// TIA Portal project "Rapid_Dyeing" (V16)
// Rapid machine for Dyeing Automation

(* hardware
DEVICE "HMI_1"  KTP400 Basic PN
   slot 0: "HMI_1"  KTP400 Basic PN  6AV2 123-2DB03-0AX0  16.0.0.0
   slot 1: "HMI_RT_1"  KTP400 Basic PN  6AV2 123-2DB03-0AX0  16.0.0.0
   slot 5: "HMI_1.IE_CP_1"  PROFINET Interface  16.0.0.0
      slot 1: "PROFINET Interface_1"  PROFINET Interface
         slot 1: "Port_1"  Port
DEVICE "S7-1200 station_1"  S7-1200 Station
   slot 0: "Rack_0"  S7-1200 Rack  Rack  V1.0
   slot 1: "PLC_1"  CPU 1212C AC/DC/Rly  6ES7 212-1BE40-0XB0  V4.4
   slot 2: "AI 4x13BIT/AQ 2x14BIT_1"  6ES7 234-4HE32-0XB0  V2.0
   slot 3: "AI 1xRTD_1"  AI1 x RTD signal board  6ES7 231-5PA30-0XB0  V2.0
*)

// ===== PLC "PLC_1"  CPU 1212C AC/DC/Rly =====

VAR_GLOBAL   // PLC tag table "Digital Inputs"
   "emergencyStop" AT %I0.0 : Bool;   // Emergency Stop Mushroom
   "faultDrive" AT %I0.2 : Bool;   // Signal from drive
   "Clock_Byte" AT %MB100 : Byte;
   "Clock_10Hz" AT %M100.0 : Bool;
   "Clock_5Hz" AT %M100.1 : Bool;
   "Clock_2.5Hz" AT %M100.2 : Bool;
   "Clock_2Hz" AT %M100.3 : Bool;
   "Clock_1.25Hz" AT %M100.4 : Bool;
   "Clock_1Hz" AT %M100.5 : Bool;
   "Clock_0.625Hz" AT %M100.6 : Bool;
   "Clock_0.5Hz" AT %M100.7 : Bool;
   "doorSensor" AT %I0.1 : Bool;   // Door sensor for safety
   "driveHandMode" AT %I0.3 : Bool;   // Selector for hand drive mode
END_VAR

VAR_GLOBAL   // PLC tag table "Digital Outputs"
   "DriveCW" AT %Q0.0 : Bool;   // Run drive ClockWise
   "DriveCCW" AT %Q0.1 : Bool;   // Run drive CounterClockWise
   "AlarmsIndicator" AT %Q0.2 : Bool;   // Alarms indicator
   "FinishedProgram" AT %Q0.3 : Bool;   // Finished program indicator
   "Heating" AT %Q0.4 : Bool;   // Heather output control
   "Cooling" AT %Q0.5 : Bool;   // Cooling output control
END_VAR

VAR_GLOBAL   // PLC tag table "Analog Inputs"
   "PT100 Feedback" AT %IW13 : Int;   // PT100 Value from process
   "feedbackFrequency" AT %IW5 : Int;
   "reserve_IN_CH1" AT %IW7 : Int;
   "reserve_IN_CH2" AT %IW9 : Int;
   "reserve_IN_CH3" AT %IW11 : Int;
END_VAR

VAR_GLOBAL   // PLC tag table "Analog Outputs"
   "frequencyOutput" AT %QW96 : Int;   // Analog output for drive frequency reference
   "reserve_Q_CH1" AT %QW98 : Int;
END_VAR

TYPE "RecipeUDT"
   STRUCT
      Frequency : Real;   // Frequency SetPoint Value
      HeatingTemperature : Real;   // Temperature SetPoint for Heating Process
      CoolingTemperature : Real;   // Temperature SetPoint for Cooling Process
      TurnTime : DInt;   // Time for Motor TurnTime
      HoldTime : DInt;   // Time for Holding Process After the SetPoint Heating Temperature is Reached
      "Gradient°C/min" : Real;   // Value for Temperature Gradient
      RecipeName : String;   // String Var for Store The Name of Current Recipe
   END_STRUCT;
END_TYPE

TYPE "TimesUDT"
   STRUCT
      Aux_Min : DInt;
      Minutes : Time;
      ElapsedTime : Time;
      Remaining : Real;
   END_STRUCT;
END_TYPE

// folder: Data

DATA_BLOCK "HMI_Vars"   // DB1
{ S7_Optimized_Access := 'TRUE' }
VERSION : 0.1
   VAR
      TechnicalService : Struct
         Inputs : Struct
            doorSensor : Bool;
         END_STRUCT;
         Outputs : Struct
            test : Bool;
         END_STRUCT;
      END_STRUCT;
      Drive : Struct
         TimeCW : Time;
         TimeCCW : Time;
         SetPoint : Real;   // Frequency SetPoint
         handAutoMode : Bool;   // Select Hand or Auto Mode
         JogCW : Bool;
         JogCCW : Bool;
         DriveCW : Bool;
         DriveCCW : Bool;
         ResetDrive : Bool;   // Reset Drive Output Signal
         HandMode : Bool;   // Hand Mode Indicator
         AutoMode : Bool;   // Auto Mode Indicator
         TurnTime_Sec : DInt;
         Run : Bool;   // Drive Run Indicator
      END_STRUCT;
      Alarms : Struct   // Reset Alarms
         Reset : Bool;
      END_STRUCT;
      runProgram : Bool;   // Run Program HMI Button
      stopProgram : Bool;   // Stop Program HMI Button
      pauseProgram : Bool;   // Pause Program HMI Button
   END_VAR
BEGIN
END_DATA_BLOCK

DATA_BLOCK "Flags"   // DB2
{ S7_Optimized_Access := 'TRUE' }
VERSION : 0.1
   VAR
      readyToStart : Bool;   // Flag for Enable All
      doorSensor : Bool;
      emergencyStop : Bool;
      faultDrive : Bool;
      finishedCooling : Bool;
      finishedRampHeating : Bool;
      runProgram : Bool;
      pauseProgram : Bool;
      startCooling : Bool;
      startTemp : Bool;
      resetPIDTemp : Bool;
      Drive : Struct
         Run : Bool;
         driveCW : Bool;
         driveCCW : Bool;
         runCW_H : Bool;
         runCCW_H : Bool;
         driveCW_H : Bool;
         driveCCW_H : Bool;
         runJogCW : Bool;
         runJogCCW : Bool;
         runCW : Bool;
         runCCW : Bool;
         AuxOutFrequency : Real;
         AuxFeedbackFrequency : Real;
         CurrentFrequency : Real;
      END_STRUCT;
   END_VAR
BEGIN
END_DATA_BLOCK

DATA_BLOCK "Temperature"   // DB4
{ S7_Optimized_Access := 'FALSE' }
VERSION : 0.1
   VAR
      "Gradient_°C/seg" : Real;   // Temperature Gradient °C/seg
      RampSetPoint : Real;   // SetPoint Output Value from Ramp Function
      ProcessValue : Real;   // Process Value Formatted
      SetPoint : Real;
   END_VAR
BEGIN
END_DATA_BLOCK

DATA_BLOCK "Alarms&Events"   // DB8
{ S7_Optimized_Access := 'FALSE' }
VERSION : 0.1
   VAR
      emergencyStop : Bool;
      doorOpen : Bool;
      faultDrive : Bool;
      finishedProgram : Bool;
   END_VAR
BEGIN
END_DATA_BLOCK

DATA_BLOCK "Recipes"   // DB9
{ S7_Optimized_Access := 'TRUE' }
VERSION : 0.1
   VAR
      RecipeVars : "RecipeUDT";
   END_VAR
BEGIN
END_DATA_BLOCK

DATA_BLOCK "JustTesting"   // DB12
{ S7_Optimized_Access := 'TRUE' }
VERSION : 0.1
   VAR
      doorsensor : Bool;
      emergencystop : Bool;
      faultdrive : Bool;
      enable : Bool;
      mode : String;
      alarmIndicator : Bool;
      Stat : Bool;
   END_VAR
BEGIN
END_DATA_BLOCK

DATA_BLOCK "Times"   // DB17
{ S7_Optimized_Access := 'TRUE' }
VERSION : 0.1
   VAR
      TotalTime_Min : Real;
      TotalTime_Remaining : Real;
      HoldTime_Remaining : Real;   // Temperature Hold Time Remaining
      AuxTurnTime_Sec : DInt;   // Turn Time Seconds
      TurnTime_Remaining : DInt;   // Turn Time Second Remaining
      Drive : Struct   // Vars for Elapsed Time and Remaining Time CW and CCW Drive Mode
         ElapsedTimeCW_TurnTime : Time;
         ElapsedTimeCCW_TurnTime : Time;
         TurnTimeCW_Remaining : Int;
         TurnTimeCCW_Remaining : Int;
         TurnTime_Sec : DInt;
      END_STRUCT;
      Heating : Struct   // Vars for Heating Ramp Time. Ramp Time Minutes and Remaining Time
         RampTime_Min : DInt;
         Remaining : Real;
      END_STRUCT;
      Cooling : Struct   // Vars for Heating Ramp Time. Ramp Time Minutes and Remaining Time
         RampTime_Min : DInt;
         Remaining : Real;
      END_STRUCT;
   END_VAR
BEGIN
END_DATA_BLOCK

// folder: Data/Block DBs

DATA_BLOCK "RTD & Gradient Value_DB"   // DB10
{ S7_Optimized_Access := 'TRUE' }
VERSION : 0.1
// stored: InstanceOfName RTD & Gradient Value
"RTD & Gradient Value"
BEGIN
END_DATA_BLOCK

DATA_BLOCK "Ramp_DB"   // DB11
{ S7_Optimized_Access := 'TRUE' }
VERSION : 0.1
// stored: InstanceOfName Ramp
"Ramp"
BEGIN
END_DATA_BLOCK

DATA_BLOCK "Process Times_DB"   // DB16
{ S7_Optimized_Access := 'TRUE' }
VERSION : 0.1
// stored: InstanceOfName Process Times
"Process Times"
BEGIN
END_DATA_BLOCK

// folder: System blocks/Program resources

DATA_BLOCK "TimeDriveCW"   // DB5
{ S7_Optimized_Access := 'TRUE' }
AUTHOR : Simatic
FAMILY : IEC
NAME : IEC_TMR
VERSION : 1.0
// stored: InstanceOfName IEC_TIMER
"IEC_TIMER"
BEGIN
END_DATA_BLOCK

DATA_BLOCK "TimeDriveCCW"   // DB6
{ S7_Optimized_Access := 'TRUE' }
AUTHOR : Simatic
FAMILY : IEC
NAME : IEC_TMR
VERSION : 1.0
// stored: InstanceOfName IEC_TIMER
"IEC_TIMER"
BEGIN
END_DATA_BLOCK

DATA_BLOCK "CoolingRampTime"   // DB13
{ S7_Optimized_Access := 'TRUE' }
AUTHOR : Simatic
FAMILY : IEC
NAME : IEC_TMR
VERSION : 1.0
// stored: InstanceOfName IEC_TIMER
"IEC_TIMER"
BEGIN
END_DATA_BLOCK

DATA_BLOCK "HeatingRampTime"   // DB14
{ S7_Optimized_Access := 'TRUE' }
AUTHOR : Simatic
FAMILY : IEC
NAME : IEC_TMR
VERSION : 1.0
// stored: InstanceOfName IEC_TIMER
"IEC_TIMER"
BEGIN
END_DATA_BLOCK

DATA_BLOCK "HoldTime"   // DB15
{ S7_Optimized_Access := 'TRUE' }
AUTHOR : Simatic
FAMILY : IEC
NAME : IEC_TMR
VERSION : 1.0
// stored: InstanceOfName IEC_TIMER
"IEC_TIMER"
BEGIN
END_DATA_BLOCK

// folder: FB

FUNCTION_BLOCK "RTD & Gradient Value"   // FB1, LAD
{ S7_Optimized_Access := 'TRUE' }
VERSION : 0.1
   VAR_INPUT
      PT100_AI : Int;   // RTD AI
      "Gradient_°C/min" : Real;   // Gradient in min from user input
   END_VAR
   VAR_OUTPUT
      ProcessValue : Real;   // Real Process Value
      "Gradient_°C/seg" : Real;   // Gradient value correct for Ramp function
   END_VAR
   VAR
      RawValue : Real;   // Raw value int to real
   END_VAR
   VAR CONSTANT
      DivRTD : Real := 10.0;   // Div input from AI pero 10.0 to give redeable value
      DivGradient : Real := 60.0;   // Div input value in min per 60.0 to give value in seg
   END_VAR
BEGIN

REGION Network 1: Convert Raw Value from AI RTD to Real redeable value.
   // e.g. RawValue 275 -> Redeable Value 27.5
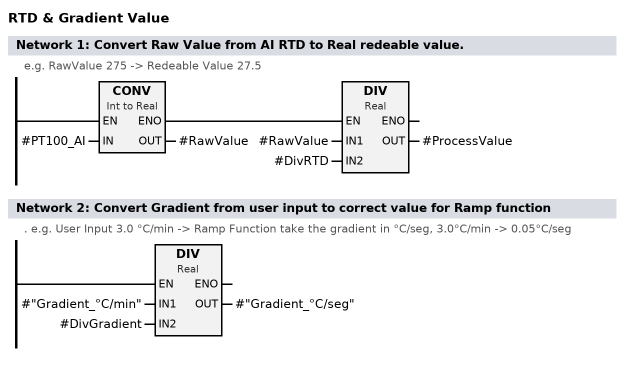
   RUNG wire#powerrail
      { S7_Templates := "[SrcType := Int, DestType := Real]" } Convert(in := #PT100_AI, out => #RawValue)
      { S7_Templates := "SrcType := Real" } Div(in1 := #RawValue, in2 := #DivRTD, out => #ProcessValue)
   END_RUNG
   // the same network as SCL:
   #RawValue := INT_TO_REAL(#PT100_AI);
   #ProcessValue := #RawValue / #DivRTD;
END_REGION

REGION Network 2: Convert Gradient from user input to correct value for Ramp function
   // . e.g. User Input 3.0 °C/min -> Ramp Function take the gradient in °C/seg, 3.0°C/min -> 0.05°C/seg
   RUNG wire#powerrail
      { S7_Templates := "SrcType := Real" } Div(in1 := #"Gradient_°C/min", in2 := #DivGradient, out => #"Gradient_°C/seg")
   END_RUNG
   // the same network as SCL:
   #"Gradient_°C/seg" := #"Gradient_°C/min" / #DivGradient;
END_REGION
END_FUNCTION_BLOCK

FUNCTION_BLOCK "Process Times"   // FB2, LAD
{ S7_Optimized_Access := 'TRUE' }
VERSION : 0.1
   VAR_INPUT
      ResetTimers : Bool;   // Reset all timers
      F_RunProgram : Bool;
      F_PauseProgram : Bool;
      HoldTime_ms : DInt;   // Time for holding Heating Temperature
      Recipe_TurnTime : DInt;
      ElapsedTimeCW_TurnTime : DInt;
      ElapsedTimeCCW_TurnTime : DInt;
      Heating_SetPoint : Real;   // Temperature Setpoint for Heating Process
      Cooling_SetPoint : Real;   // Temperature SetPoint for Cooling Process
      Temp_ProcessValue : Real;   // Temperature Process Value
      StartTemp : Real;
      TempGradient : Real;   // Temperature gradient
   END_VAR
   VAR_OUTPUT
      HoldTime_Remaining : Real;
      TurnTimeCW_Remaining : Int;
      TurnTimeCCW_Remaining : Int;
      HeatingRampTime_Min : Real;
      CoolingRampTime_Min : Real;
      TotalTime_Min : Real;
      TotalTime_Remaining : Real;
      Heating_Remaining : Real;
      Cooling_Remaining : Real;
      F_FinishedHoldTimeOut : Bool;   // Signal for finish time. Hold time heating temperature
      F_FinishedCoolingOut : Bool;
      F_FinishedRampHeating : Bool;
      DriveTurnTime_Sec : Time;
   END_VAR
   VAR
      HoldTime : Struct
         HoldTime_ms : DInt;
         Minutes : Time;
         ElapsedTime : Time;
         Remaining : Real;
         Total : DInt;
      END_STRUCT;
      Drive : Struct
         AuxRemCW : Int;
         AuxRemCCW : Int;
         AuxTurnTime_Sec : Int;
         TurnTime_Sec : Time;
         Remaining : DInt;
      END_STRUCT;
      Heating : Struct
         AuxSpan : Real;
         Ramp_min : Real;
         Ramp_ms : Real;
         Ramp_time_ms : Time;
         ElapsedTime : DInt;
         Remaining : Real;
      END_STRUCT;
      Cooling : Struct
         AuxSpan : Real;
         Ramp_min : Real;
         Ramp_ms : Real;
         Ramp_time_ms : Time;
         ElapsedTime : DInt;
         Remaining : Real;
      END_STRUCT;
   END_VAR
   VAR CONSTANT
      "ms to min" : DInt := 60000;
      "ms to sec" : DInt := 1000;
      HighTemp : Real := 127.0;
      LowTemp : Real := 130.0;
   END_VAR
BEGIN

REGION Network 1: Formatting values of Hold Time
   // 1st. Convert ms from recipe var to minutes
   // 2nd. Pass the minutes to PT timer
   // 3rd. Sub. PT - ET for obtain the remaining time in ms. Finally Div the ms to obtain remaining time in minutes.
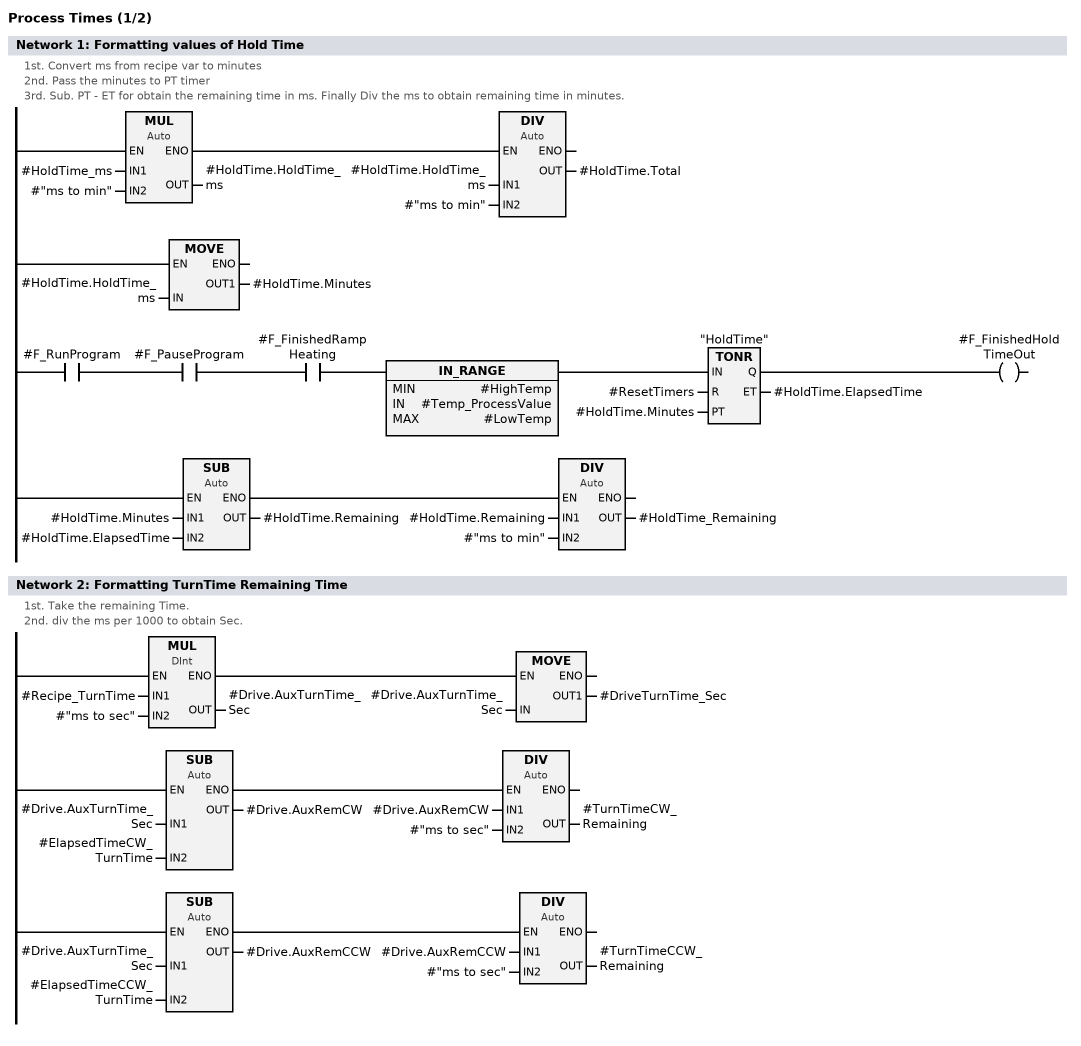
   #HoldTime.HoldTime_ms := #HoldTime_ms * #"ms to min";
   #HoldTime.Total := #HoldTime.HoldTime_ms / #"ms to min";
   #HoldTime.Minutes := #HoldTime.HoldTime_ms;
   "HoldTime".TONR(IN := #F_RunProgram AND #F_PauseProgram AND #F_FinishedRampHeating AND (#HighTemp <= #Temp_ProcessValue) AND (#Temp_ProcessValue <= #LowTemp),
                   R := #ResetTimers,
                   PT := #HoldTime.Minutes,
                   ET => #HoldTime.ElapsedTime);
   #F_FinishedHoldTimeOut := "HoldTime".Q;
   #HoldTime.Remaining := #HoldTime.Minutes - #HoldTime.ElapsedTime;
   #HoldTime_Remaining := #HoldTime.Remaining / #"ms to min";
END_REGION

REGION Network 2: Formatting TurnTime Remaining Time
   // 1st. Take the remaining Time.
   // 2nd. div the ms per 1000 to obtain Sec.
   RUNG wire#powerrail
      { S7_Templates := "SrcType := DInt" } Mul(in1 := #Recipe_TurnTime, in2 := #"ms to sec", out => #Drive.AuxTurnTime_Sec)
      Move(in := #Drive.AuxTurnTime_Sec, out1 => #DriveTurnTime_Sec)
   END_RUNG
   RUNG wire#powerrail
      Sub(in1 := #Drive.AuxTurnTime_Sec, in2 := #ElapsedTimeCW_TurnTime, out => #Drive.AuxRemCW)
      Div(in1 := #Drive.AuxRemCW, in2 := #"ms to sec", out => #TurnTimeCW_Remaining)
   END_RUNG
   RUNG wire#powerrail
      Sub(in1 := #Drive.AuxTurnTime_Sec, in2 := #ElapsedTimeCCW_TurnTime, out => #Drive.AuxRemCCW)
      Div(in1 := #Drive.AuxRemCCW, in2 := #"ms to sec", out => #TurnTimeCCW_Remaining)
   END_RUNG
   // the same network as SCL:
   #Drive.AuxTurnTime_Sec := #Recipe_TurnTime * #"ms to sec";
   #DriveTurnTime_Sec := #Drive.AuxTurnTime_Sec;
   #Drive.AuxRemCW := #Drive.AuxTurnTime_Sec - #ElapsedTimeCW_TurnTime;
   #TurnTimeCW_Remaining := #Drive.AuxRemCW / #"ms to sec";
   #Drive.AuxRemCCW := #Drive.AuxTurnTime_Sec - #ElapsedTimeCCW_TurnTime;
   #TurnTimeCCW_Remaining := #Drive.AuxRemCCW / #"ms to sec";
END_REGION

REGION Network 3: Calculate Ramp Heating Time and Remaining Time
   // Formula
   // ΔT = T_Set - T_Actual (SPAN)
   // Time_min = ΔT / 3.0
   // Time_ms = Time_min * 60000
   // 
   // The T_Actual is equal to Cooling Temperature that is where start process and finished process.
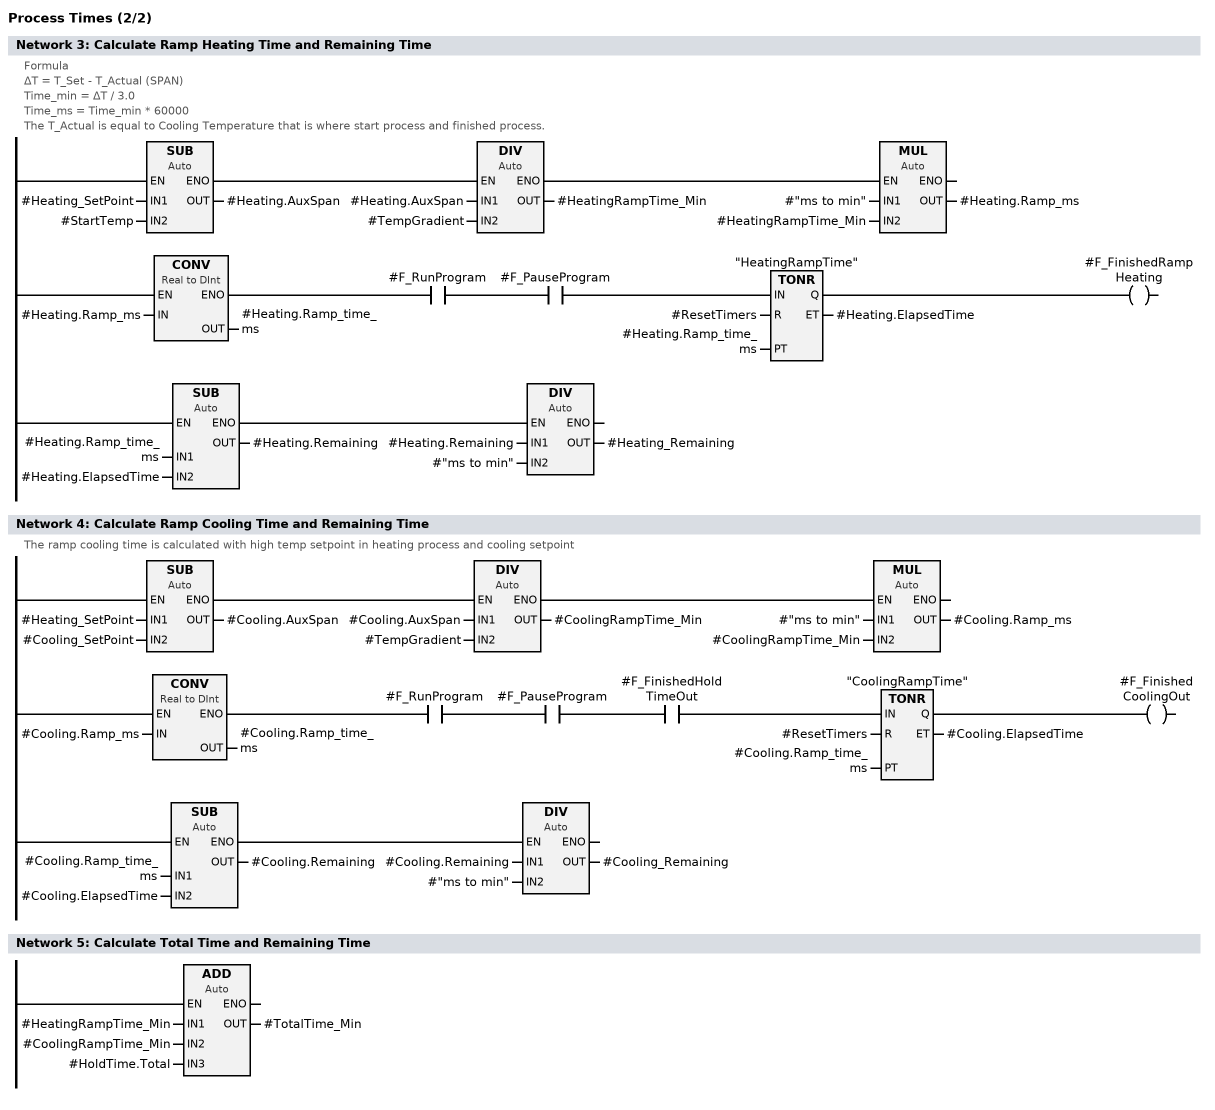
   #Heating.AuxSpan := #Heating_SetPoint - #StartTemp;
   #HeatingRampTime_Min := #Heating.AuxSpan / #TempGradient;
   #Heating.Ramp_ms := #"ms to min" * #HeatingRampTime_Min;
   #Heating.Ramp_time_ms := REAL_TO_DINT(#Heating.Ramp_ms);
   "HeatingRampTime".TONR(IN := #F_RunProgram AND #F_PauseProgram,
                          R := #ResetTimers,
                          PT := #Heating.Ramp_time_ms,
                          ET => #Heating.ElapsedTime);
   #F_FinishedRampHeating := "HeatingRampTime".Q;
   #Heating.Remaining := #Heating.Ramp_time_ms - #Heating.ElapsedTime;
   #Heating_Remaining := #Heating.Remaining / #"ms to min";
END_REGION

REGION Network 4: Calculate Ramp Cooling Time and Remaining Time
   // The ramp cooling time is calculated with high temp setpoint in heating process and cooling setpoint
   #Cooling.AuxSpan := #Heating_SetPoint - #Cooling_SetPoint;
   #CoolingRampTime_Min := #Cooling.AuxSpan / #TempGradient;
   #Cooling.Ramp_ms := #"ms to min" * #CoolingRampTime_Min;
   #Cooling.Ramp_time_ms := REAL_TO_DINT(#Cooling.Ramp_ms);
   "CoolingRampTime".TONR(IN := #F_RunProgram AND #F_PauseProgram AND #F_FinishedHoldTimeOut,
                          R := #ResetTimers,
                          PT := #Cooling.Ramp_time_ms,
                          ET => #Cooling.ElapsedTime);
   #F_FinishedCoolingOut := "CoolingRampTime".Q;
   #Cooling.Remaining := #Cooling.Ramp_time_ms - #Cooling.ElapsedTime;
   #Cooling_Remaining := #Cooling.Remaining / #"ms to min";
END_REGION

REGION Network 5: Calculate Total Time and Remaining Time
   RUNG wire#powerrail
      Add(in1 := #HeatingRampTime_Min, in2 := #CoolingRampTime_Min, in3 := #HoldTime.Total, out => #TotalTime_Min)
   END_RUNG
   // the same network as SCL:
   #TotalTime_Min := #HeatingRampTime_Min + #CoolingRampTime_Min + #HoldTime.Total;
END_REGION
END_FUNCTION_BLOCK

FUNCTION_BLOCK "Ramp"   // FB3, SCL
{ S7_Optimized_Access := 'TRUE' }
VERSION : 0.1
   VAR_INPUT
      InitFB : Bool;
      SetPoint : Real;
      Rate : Real;
   END_VAR
   VAR_OUTPUT
      Out : Real;
   END_VAR
   VAR
      ActualTime : DTL;
      LastTime : DTL;
      AuxOut : Real;
   END_VAR
   VAR_TEMP
      DeltaTime_T : Time;
      DeltaTime_DI : DInt;
      DeltaTime : Real;
      auxR : Real;
      auxDI : DInt;
      rv1 : Int;
   END_VAR
BEGIN
   #rv1:= RD_SYS_T(#ActualTime);

   IF #InitFB = true THEN
       #LastTime := #ActualTime;
       #AuxOut := #SetPoint;
       #Out := #AuxOut;
   END_IF;

   #DeltaTime_T:= T_DIFF(IN1:=#ActualTime, IN2:=#LastTime);
   #DeltaTime_DI:= TIME_TO_DINT(#DeltaTime_T);
   #DeltaTime:= DINT_TO_REAL(#DeltaTime_DI);
   #DeltaTime := #DeltaTime / 1000.0;
   #LastTime := #ActualTime;

   IF #SetPoint < #AuxOut THEN
       #Out := #AuxOut;
       #auxR := #AuxOut - (#Rate * #DeltaTime);
       #Out := #AuxOut;
       #AuxOut := MAX(IN1 := #auxR, IN2 := #SetPoint);
       #Out := #AuxOut;
       RETURN;
   ELSE
       IF #SetPoint > #AuxOut THEN
           #Out := #AuxOut;
           #auxR := (#Rate * #DeltaTime) + #AuxOut;
           #Out := #AuxOut;
           #AuxOut := MIN(IN1 := #auxR, IN2 := #SetPoint);
           #Out := #AuxOut;
       END_IF;
   END_IF;
   RETURN;
END_FUNCTION_BLOCK

// folder: FC

FUNCTION "Initial Conditions" : Void   // FC1, LAD
{ S7_Optimized_Access := 'TRUE' }
VERSION : 0.1
   VAR_INPUT
      EmergencyStop : Bool;
      HMIRunProgram : Bool;
      HMIPauseProgram : Bool;
      HMIStopProgram : Bool;
      FaultDrive : Bool;
   END_VAR
   VAR_OUTPUT
      F_RunProgram : Bool;
      F_PauseProgram : Bool;
   END_VAR
   VAR_IN_OUT
      F_ReadyToStart : Bool;
      F_EmergencyStop : Bool;
      F_FaultDrive : Bool;
   END_VAR
BEGIN

REGION Network 1: Flags
   // Enable program when selector switch is change to 1
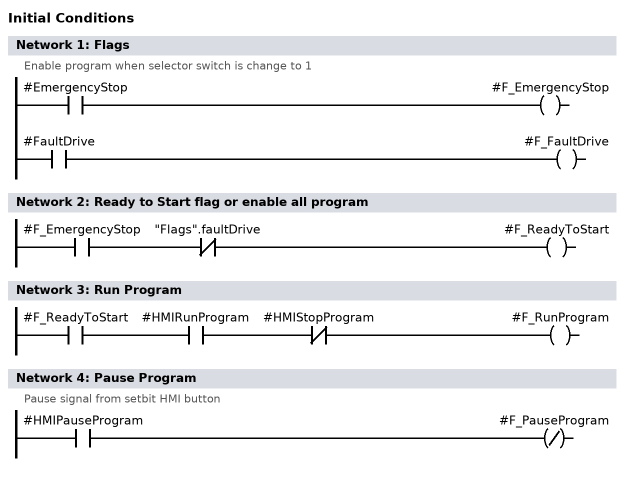
   RUNG wire#powerrail
      Contact( #EmergencyStop )
      Coil( #F_EmergencyStop )
   END_RUNG
   RUNG wire#powerrail
      Contact( #FaultDrive )
      Coil( #F_FaultDrive )
   END_RUNG
   // the same network as SCL:
   #F_EmergencyStop := #EmergencyStop;
   #F_FaultDrive := #FaultDrive;
END_REGION

REGION Network 2: Ready to Start flag or enable all program
   RUNG wire#powerrail
      Contact( #F_EmergencyStop )
      I_Contact( "Flags".faultDrive )
      Coil( #F_ReadyToStart )
   END_RUNG
   // the same network as SCL:
   #F_ReadyToStart := #F_EmergencyStop AND NOT "Flags".faultDrive;
END_REGION

REGION Network 3: Run Program
   RUNG wire#powerrail
      Contact( #F_ReadyToStart )
      Contact( #HMIRunProgram )
      I_Contact( #HMIStopProgram )
      Coil( #F_RunProgram )
   END_RUNG
   // the same network as SCL:
   #F_RunProgram := #F_ReadyToStart AND #HMIRunProgram AND NOT #HMIStopProgram;
END_REGION

REGION Network 4: Pause Program
   // Pause signal from setbit HMI button
   RUNG wire#powerrail
      Contact( #HMIPauseProgram )
      I_Coil( #F_PauseProgram )
   END_RUNG
   // the same network as SCL:
   #F_PauseProgram := NOT #HMIPauseProgram;
END_REGION
END_FUNCTION

FUNCTION "Drive Control" : Void   // FC2, LAD
TITLE = Logic for Controlling Drive in Hand or Auto Mode
{ S7_Optimized_Access := 'TRUE' }
VERSION : 0.1
   VAR_INPUT
      F_ReadytoStart : Bool;
      handAutoMode : Bool;
      HMIDriveCW : Bool;
      HMIDriveCCW : Bool;
      DoorSensor : Bool;
      F_RunProgram : Bool;
      F_PauseProgram : Bool;
      TurnTime : Time;
      FeedbackFrequency : Real;
      RecipeFrequency : Real;
      HandFrequency : Real;
   END_VAR
   VAR_OUTPUT
      DriveCW : Bool;
      DriveCCW : Bool;
      Run : Bool;
      OutputFrequency : Int;
      CurrentFrequency : Real;
   END_VAR
   VAR_IN_OUT
      AutoMode : Bool;
      F_DoorSensor : Bool;
      HandMode : Bool;
      F_DriveCW : Bool;
      F_DriveCCW : Bool;
      F_DriveRunCW : Bool;
      F_DriveRunCCW : Bool;
      F_DriveCW_H : Bool;
      F_DriveCCW_H : Bool;
      F_DriveRunCW_H : Bool;
      F_DriveRunCCW_H : Bool;
      ElapsedTimeCW_TurnTime : Time;
      ElapsedTimeCCW_TurnTime : Time;
      AuxOutFrequency : Real;
      AuxFeedbackFrequency : Real;
      FrequencySetPoint : Real;
   END_VAR
   VAR CONSTANT
      msToSec : DInt := 1000;
      Min_Hz : Real := 0.0;
      Max_Hz : Real := 60.0;
      Min_Analog : Int := 0;
      Max_Analog : Int := 27648;
   END_VAR
   VAR_TEMP   // added for the SCL form of the ladder/FBD networks
      _w1 : Bool;
   END_VAR
BEGIN

REGION Network 1: Door Sensor Flag
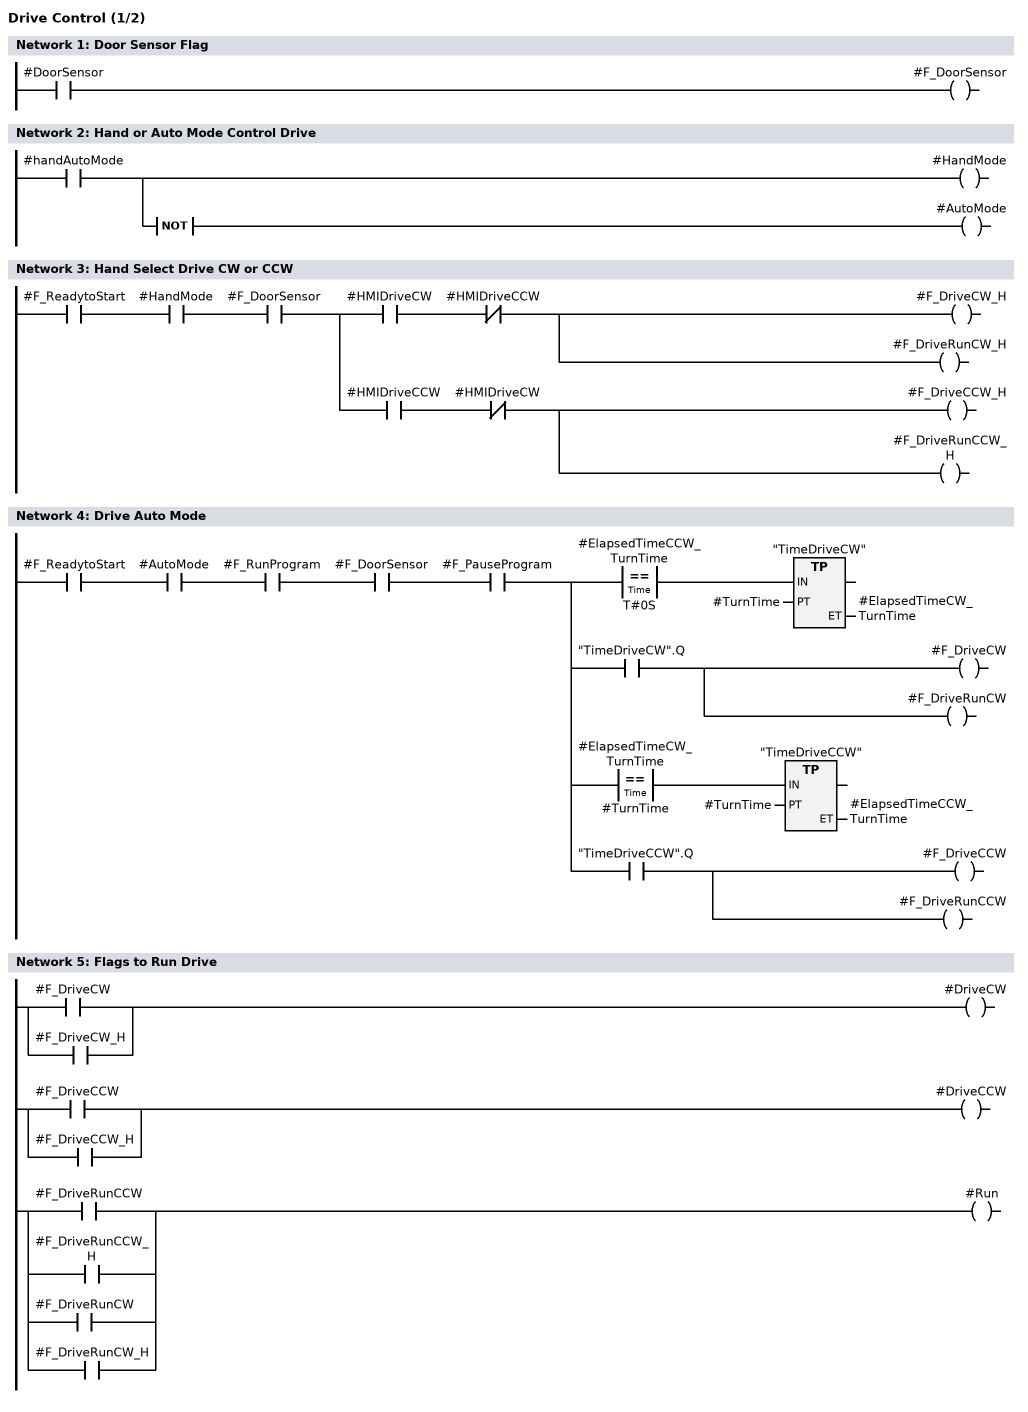
   RUNG wire#powerrail
      Contact( #DoorSensor )
      Coil( #F_DoorSensor )
   END_RUNG
   // the same network as SCL:
   #F_DoorSensor := #DoorSensor;
END_REGION

REGION Network 2: Hand or Auto Mode Control Drive
   RUNG wire#powerrail
      Contact( #handAutoMode )
      wire#w1
      Coil( #HandMode )
   END_RUNG
   RUNG wire#w1
      Not()
      Coil( #AutoMode )
   END_RUNG
   // the same network as SCL:
   #HandMode := #handAutoMode;
   #AutoMode := NOT #handAutoMode;
END_REGION

REGION Network 3: Hand Select Drive CW or CCW
   RUNG wire#powerrail
      Contact( #F_ReadytoStart )
      Contact( #HandMode )
      Contact( #F_DoorSensor )
      wire#w1
      Contact( #HMIDriveCW )
      I_Contact( #HMIDriveCCW )
      wire#w2
      Coil( #F_DriveCW_H )
   END_RUNG
   RUNG wire#w2
      Coil( #F_DriveRunCW_H )
   END_RUNG
   RUNG wire#w1
      Contact( #HMIDriveCCW )
      I_Contact( #HMIDriveCW )
      wire#w3
      Coil( #F_DriveCCW_H )
   END_RUNG
   RUNG wire#w3
      Coil( #F_DriveRunCCW_H )
   END_RUNG
   // the same network as SCL:
   #_w1 := #F_ReadytoStart AND #HandMode AND #F_DoorSensor;
   #F_DriveCW_H := #_w1 AND #HMIDriveCW AND NOT #HMIDriveCCW;
   #F_DriveRunCW_H := #F_DriveCW_H;
   #F_DriveCCW_H := #_w1 AND #HMIDriveCCW AND NOT #HMIDriveCW;
   #F_DriveRunCCW_H := #F_DriveCCW_H;
END_REGION

REGION Network 4: Drive Auto Mode
   #_w1 := #F_ReadytoStart AND #AutoMode AND #F_RunProgram AND #F_DoorSensor AND #F_PauseProgram;
   "TimeDriveCW".TP(IN := #_w1 AND (#ElapsedTimeCCW_TurnTime = T#0S),
                    PT := #TurnTime,
                    ET => #ElapsedTimeCW_TurnTime);
   #F_DriveCW := #_w1 AND "TimeDriveCW".Q;
   #F_DriveRunCW := #F_DriveCW;
   "TimeDriveCCW".TP(IN := #_w1 AND (#ElapsedTimeCW_TurnTime = #TurnTime),
                     PT := #TurnTime,
                     ET => #ElapsedTimeCCW_TurnTime);
   #F_DriveCCW := #_w1 AND "TimeDriveCCW".Q;
   #F_DriveRunCCW := #F_DriveCCW;
END_REGION

REGION Network 5: Flags to Run Drive
   RUNG wire#powerrail
      Contact( #F_DriveCW )
      wire#w1
      Coil( #DriveCW )
   END_RUNG
   RUNG wire#powerrail
      Contact( #F_DriveCW_H )
   END_RUNG wire#w1
   RUNG wire#powerrail
      Contact( #F_DriveCCW )
      wire#w2
      Coil( #DriveCCW )
   END_RUNG
   RUNG wire#powerrail
      Contact( #F_DriveCCW_H )
   END_RUNG wire#w2
   RUNG wire#powerrail
      Contact( #F_DriveRunCCW )
      wire#w3
      Coil( #Run )
   END_RUNG
   RUNG wire#powerrail
      Contact( #F_DriveRunCCW_H )
   END_RUNG wire#w3
   RUNG wire#powerrail
      Contact( #F_DriveRunCW )
   END_RUNG wire#w3
   RUNG wire#powerrail
      Contact( #F_DriveRunCW_H )
   END_RUNG wire#w3
   // the same network as SCL:
   #DriveCW := #F_DriveCW OR #F_DriveCW_H;
   #DriveCCW := #F_DriveCCW OR #F_DriveCCW_H;
   #Run := #F_DriveRunCCW OR #F_DriveRunCCW_H OR #F_DriveRunCW OR #F_DriveRunCW_H;
END_REGION

REGION Network 6: Output Frequency Control
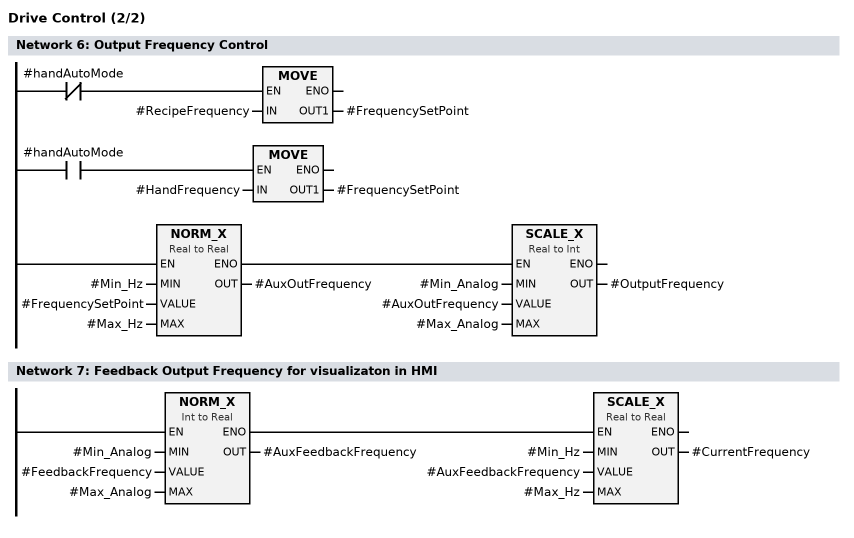
   RUNG wire#powerrail
      I_Contact( #handAutoMode )
      Move(in := #RecipeFrequency, out1 => #FrequencySetPoint)
   END_RUNG
   RUNG wire#powerrail
      Contact( #handAutoMode )
      Move(in := #HandFrequency, out1 => #FrequencySetPoint)
   END_RUNG
   RUNG wire#powerrail
      { S7_Templates := "[SrcType := Real, DestType := Real]" } Normalize(min := #Min_Hz, value := #FrequencySetPoint, max := #Max_Hz, out => #AuxOutFrequency)
      { S7_Templates := "[SrcType := Real, DestType := Int]" } Scale(min := #Min_Analog, value := #AuxOutFrequency, max := #Max_Analog, out => #OutputFrequency)
   END_RUNG
   // the same network as SCL:
   IF NOT #handAutoMode THEN #FrequencySetPoint := #RecipeFrequency; END_IF;
   IF #handAutoMode THEN #FrequencySetPoint := #HandFrequency; END_IF;
   #AuxOutFrequency := NORM_X(MIN := #Min_Hz, VALUE := #FrequencySetPoint, MAX := #Max_Hz);
   #OutputFrequency := SCALE_X(MIN := #Min_Analog, VALUE := #AuxOutFrequency, MAX := #Max_Analog);
END_REGION

REGION Network 7: Feedback Output Frequency for visualizaton in HMI
   RUNG wire#powerrail
      { S7_Templates := "[SrcType := Int, DestType := Real]" } Normalize(min := #Min_Analog, value := #FeedbackFrequency, max := #Max_Analog, out => #AuxFeedbackFrequency)
      { S7_Templates := "[SrcType := Real, DestType := Real]" } Scale(min := #Min_Hz, value := #AuxFeedbackFrequency, max := #Max_Hz, out => #CurrentFrequency)
   END_RUNG
   // the same network as SCL:
   #AuxFeedbackFrequency := NORM_X(MIN := #Min_Analog, VALUE := #FeedbackFrequency, MAX := #Max_Analog);
   #CurrentFrequency := SCALE_X(MIN := #Min_Hz, VALUE := #AuxFeedbackFrequency, MAX := #Max_Hz);
END_REGION
END_FUNCTION

FUNCTION "Alarms & Events" : Void   // FC3, LAD
{ S7_Optimized_Access := 'TRUE' }
VERSION : 0.1
   VAR_INPUT
      ResetAlarms : Bool;
      F_EmergencyStop : Bool;
      F_DoorSensor : Bool;
      F_FaultDrive : Bool;
      F_FinishedProcess : Bool;
   END_VAR
   VAR_OUTPUT
      AlarmIndicator : Bool;
      FinishedProgramIndicator : Bool;
   END_VAR
   VAR_IN_OUT
      Alm_EmergencyStop : Bool;
      Alm_DoorOpen : Bool;
      Alm_FaultDrive : Bool;
      Event_FinishedProcess : Bool;
   END_VAR
BEGIN

REGION Network 1: Emergency Stop Activated
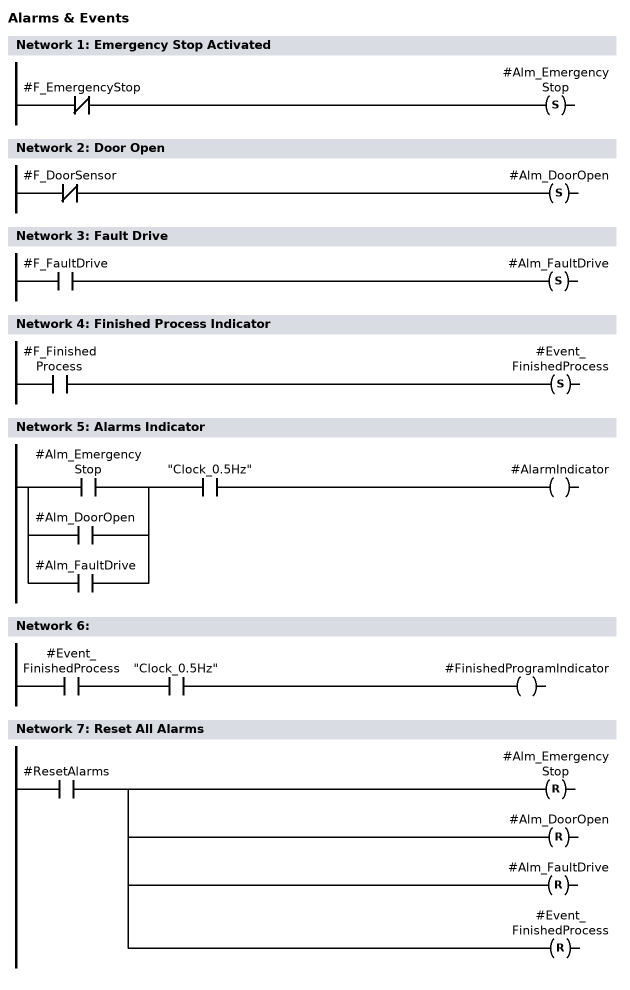
   RUNG wire#powerrail
      I_Contact( #F_EmergencyStop )
      S_Coil( #Alm_EmergencyStop )
   END_RUNG
   // the same network as SCL:
   IF NOT #F_EmergencyStop THEN #Alm_EmergencyStop := TRUE; END_IF;
END_REGION

REGION Network 2: Door Open
   RUNG wire#powerrail
      I_Contact( #F_DoorSensor )
      S_Coil( #Alm_DoorOpen )
   END_RUNG
   // the same network as SCL:
   IF NOT #F_DoorSensor THEN #Alm_DoorOpen := TRUE; END_IF;
END_REGION

REGION Network 3: Fault Drive
   RUNG wire#powerrail
      Contact( #F_FaultDrive )
      S_Coil( #Alm_FaultDrive )
   END_RUNG
   // the same network as SCL:
   IF #F_FaultDrive THEN #Alm_FaultDrive := TRUE; END_IF;
END_REGION

REGION Network 4: Finished Process Indicator
   RUNG wire#powerrail
      Contact( #F_FinishedProcess )
      S_Coil( #Event_FinishedProcess )
   END_RUNG
   // the same network as SCL:
   IF #F_FinishedProcess THEN #Event_FinishedProcess := TRUE; END_IF;
END_REGION

REGION Network 5: Alarms Indicator
   RUNG wire#powerrail
      Contact( #Alm_EmergencyStop )
      wire#w1
      Contact( "Clock_0.5Hz" )
      Coil( #AlarmIndicator )
   END_RUNG
   RUNG wire#powerrail
      Contact( #Alm_DoorOpen )
   END_RUNG wire#w1
   RUNG wire#powerrail
      Contact( #Alm_FaultDrive )
   END_RUNG wire#w1
   // the same network as SCL:
   #AlarmIndicator := (#Alm_EmergencyStop OR #Alm_DoorOpen OR #Alm_FaultDrive) AND "Clock_0.5Hz";
END_REGION

REGION Network 6
   RUNG wire#powerrail
      Contact( #Event_FinishedProcess )
      Contact( "Clock_0.5Hz" )
      Coil( #FinishedProgramIndicator )
   END_RUNG
   // the same network as SCL:
   #FinishedProgramIndicator := #Event_FinishedProcess AND "Clock_0.5Hz";
END_REGION

REGION Network 7: Reset All Alarms
   RUNG wire#powerrail
      Contact( #ResetAlarms )
      wire#w1
      R_Coil( #Alm_EmergencyStop )
   END_RUNG
   RUNG wire#w1
      R_Coil( #Alm_DoorOpen )
   END_RUNG
   RUNG wire#w1
      R_Coil( #Alm_FaultDrive )
   END_RUNG
   RUNG wire#w1
      R_Coil( #Event_FinishedProcess )
   END_RUNG
   // the same network as SCL:
   IF #ResetAlarms THEN
       #Alm_EmergencyStop := FALSE;
       #Alm_DoorOpen := FALSE;
       #Alm_FaultDrive := FALSE;
       #Event_FinishedProcess := FALSE;
   END_IF;
END_REGION
END_FUNCTION

FUNCTION "Heating & Cooling" : Void   // FC4, LAD
{ S7_Optimized_Access := 'TRUE' }
VERSION : 0.1
   VAR_INPUT
      HeatingTemperature : Real;
      CoolingTemperature : Real;
      StartHeating : Bool;
      StartCooling : Bool;
      Temp_ProcessValue : Real;
      Temp_RampSetPoint : Real;
      Temp_SetPoint : Real;
   END_VAR
   VAR_OUTPUT
      TemperatureSetPoint : Real;
      F_EnableStartTemp : Bool;
   END_VAR
   VAR CONSTANT
      StartTemp : Real := 30.0;
   END_VAR
BEGIN

REGION Network 1: Setting SetPoint depend on which process is selected
   // Start heating is selected when the run program is active.
   // Start cooling is selected when the holdtime is reached
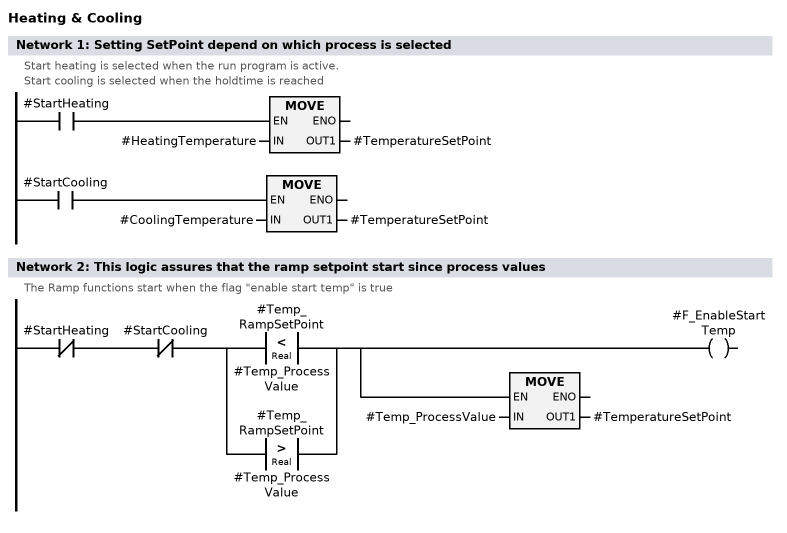
   RUNG wire#powerrail
      Contact( #StartHeating )
      Move(in := #HeatingTemperature, out1 => #TemperatureSetPoint)
   END_RUNG
   RUNG wire#powerrail
      Contact( #StartCooling )
      Move(in := #CoolingTemperature, out1 => #TemperatureSetPoint)
   END_RUNG
   // the same network as SCL:
   IF #StartHeating THEN #TemperatureSetPoint := #HeatingTemperature; END_IF;
   IF #StartCooling THEN #TemperatureSetPoint := #CoolingTemperature; END_IF;
END_REGION

REGION Network 2: This logic assures that the ramp setpoint start since process values
   // The Ramp functions start when the flag "enable start temp" is true
   RUNG wire#powerrail
      I_Contact( #StartHeating )
      I_Contact( #StartCooling )
      wire#w1
      { S7_Templates := "SrcType := Real" } LT_Contact(in1 := #Temp_RampSetPoint, in2 := #Temp_ProcessValue)
      wire#w2
      Coil( #F_EnableStartTemp )
   END_RUNG
   RUNG wire#w1
      { S7_Templates := "SrcType := Real" } GT_Contact(in1 := #Temp_RampSetPoint, in2 := #Temp_ProcessValue)
   END_RUNG wire#w2
   RUNG wire#w2
      Move(in := #Temp_ProcessValue, out1 => #TemperatureSetPoint)
   END_RUNG
   // the same network as SCL:
   #F_EnableStartTemp := NOT #StartHeating AND NOT #StartCooling AND ((#Temp_RampSetPoint < #Temp_ProcessValue) OR (#Temp_RampSetPoint > #Temp_ProcessValue));
   IF #F_EnableStartTemp THEN #TemperatureSetPoint := #Temp_ProcessValue; END_IF;
END_REGION
END_FUNCTION

// folder: Organization Blocks

ORGANIZATION_BLOCK "Main"   // OB1, LAD, ProgramCycle
TITLE = "Main Program Sweep (Cycle)"
{ S7_Optimized_Access := 'TRUE' }
VERSION : 0.1
   VAR_INPUT
      Initial_Call : Bool;   // Initial call of this OB
      Remanence : Bool;   // =True, if remanent data are available
   END_VAR
BEGIN

REGION Network 1: Initial Conditions to Run Program
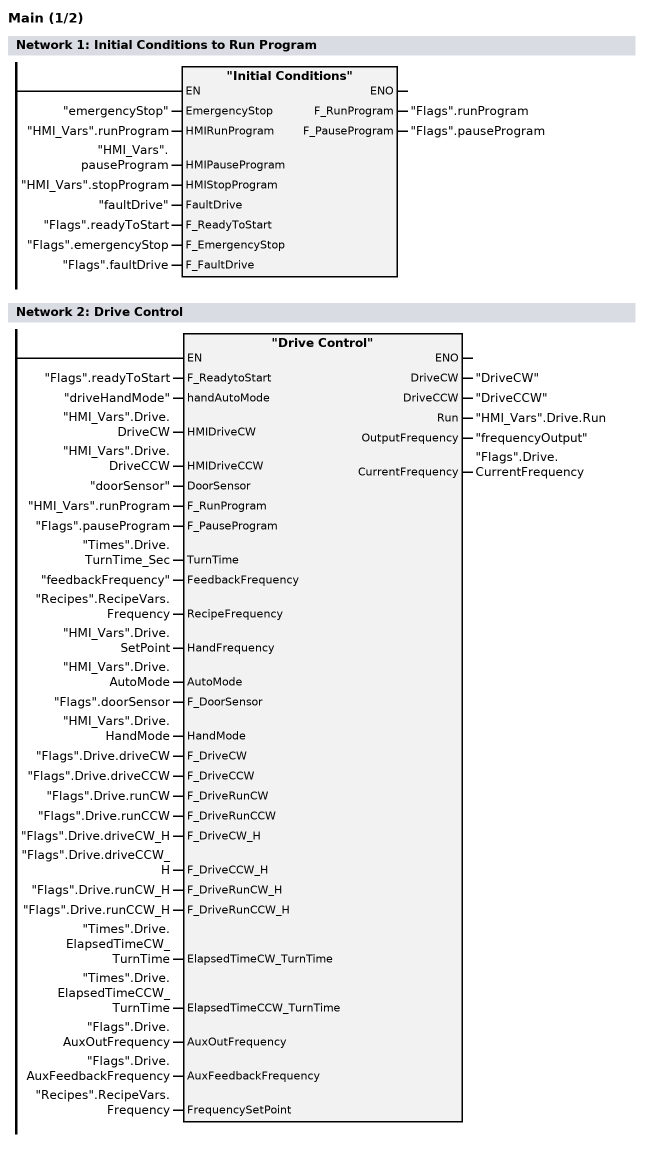
   RUNG wire#powerrail
      "Initial Conditions"(EmergencyStop := "emergencyStop", HMIRunProgram := "HMI_Vars".runProgram, HMIPauseProgram := "HMI_Vars".pauseProgram, HMIStopProgram := "HMI_Vars".stopProgram, FaultDrive := "faultDrive", F_ReadyToStart := "Flags".readyToStart, F_EmergencyStop := "Flags".emergencyStop, F_FaultDrive := "Flags".faultDrive, F_RunProgram => "Flags".runProgram, F_PauseProgram => "Flags".pauseProgram)
   END_RUNG
   // the same network as SCL:
   "Initial Conditions"(EmergencyStop := "emergencyStop",
                        HMIRunProgram := "HMI_Vars".runProgram,
                        HMIPauseProgram := "HMI_Vars".pauseProgram,
                        HMIStopProgram := "HMI_Vars".stopProgram,
                        FaultDrive := "faultDrive",
                        F_ReadyToStart := "Flags".readyToStart,
                        F_EmergencyStop := "Flags".emergencyStop,
                        F_FaultDrive := "Flags".faultDrive,
                        F_RunProgram => "Flags".runProgram,
                        F_PauseProgram => "Flags".pauseProgram);
END_REGION

REGION Network 2: Drive Control
   RUNG wire#powerrail
      "Drive Control"(F_ReadytoStart := "Flags".readyToStart, handAutoMode := "driveHandMode", HMIDriveCW := "HMI_Vars".Drive.DriveCW, HMIDriveCCW := "HMI_Vars".Drive.DriveCCW, DoorSensor := "doorSensor", F_RunProgram := "HMI_Vars".runProgram, F_PauseProgram := "Flags".pauseProgram, TurnTime := "Times".Drive.TurnTime_Sec, FeedbackFrequency := "feedbackFrequency", RecipeFrequency := "Recipes".RecipeVars.Frequency, HandFrequency := "HMI_Vars".Drive.SetPoint, AutoMode := "HMI_Vars".Drive.AutoMode, F_DoorSensor := "Flags".doorSensor, HandMode := "HMI_Vars".Drive.HandMode, F_DriveCW := "Flags".Drive.driveCW, F_DriveCCW := "Flags".Drive.driveCCW, F_DriveRunCW := "Flags".Drive.runCW, F_DriveRunCCW := "Flags".Drive.runCCW, F_DriveCW_H := "Flags".Drive.driveCW_H, F_DriveCCW_H := "Flags".Drive.driveCCW_H, F_DriveRunCW_H := "Flags".Drive.runCW_H, F_DriveRunCCW_H := "Flags".Drive.runCCW_H, ElapsedTimeCW_TurnTime := "Times".Drive.ElapsedTimeCW_TurnTime, ElapsedTimeCCW_TurnTime := "Times".Drive.ElapsedTimeCCW_TurnTime, AuxOutFrequency := "Flags".Drive.AuxOutFrequency, AuxFeedbackFrequency := "Flags".Drive.AuxFeedbackFrequency, FrequencySetPoint := "Recipes".RecipeVars.Frequency, DriveCW => "DriveCW", DriveCCW => "DriveCCW", Run => "HMI_Vars".Drive.Run, OutputFrequency => "frequencyOutput", CurrentFrequency => "Flags".Drive.CurrentFrequency)
   END_RUNG
   // the same network as SCL:
   "Drive Control"(F_ReadytoStart := "Flags".readyToStart,
                   handAutoMode := "driveHandMode",
                   HMIDriveCW := "HMI_Vars".Drive.DriveCW,
                   HMIDriveCCW := "HMI_Vars".Drive.DriveCCW,
                   DoorSensor := "doorSensor",
                   F_RunProgram := "HMI_Vars".runProgram,
                   F_PauseProgram := "Flags".pauseProgram,
                   TurnTime := "Times".Drive.TurnTime_Sec,
                   FeedbackFrequency := "feedbackFrequency",
                   RecipeFrequency := "Recipes".RecipeVars.Frequency,
                   HandFrequency := "HMI_Vars".Drive.SetPoint,
                   AutoMode := "HMI_Vars".Drive.AutoMode,
                   F_DoorSensor := "Flags".doorSensor,
                   HandMode := "HMI_Vars".Drive.HandMode,
                   F_DriveCW := "Flags".Drive.driveCW,
                   F_DriveCCW := "Flags".Drive.driveCCW,
                   F_DriveRunCW := "Flags".Drive.runCW,
                   F_DriveRunCCW := "Flags".Drive.runCCW,
                   F_DriveCW_H := "Flags".Drive.driveCW_H,
                   F_DriveCCW_H := "Flags".Drive.driveCCW_H,
                   F_DriveRunCW_H := "Flags".Drive.runCW_H,
                   F_DriveRunCCW_H := "Flags".Drive.runCCW_H,
                   ElapsedTimeCW_TurnTime := "Times".Drive.ElapsedTimeCW_TurnTime,
                   ElapsedTimeCCW_TurnTime := "Times".Drive.ElapsedTimeCCW_TurnTime,
                   AuxOutFrequency := "Flags".Drive.AuxOutFrequency,
                   AuxFeedbackFrequency := "Flags".Drive.AuxFeedbackFrequency,
                   FrequencySetPoint := "Recipes".RecipeVars.Frequency,
                   DriveCW => "DriveCW",
                   DriveCCW => "DriveCCW",
                   Run => "HMI_Vars".Drive.Run,
                   OutputFrequency => "frequencyOutput",
                   CurrentFrequency => "Flags".Drive.CurrentFrequency);
END_REGION

REGION Network 3: Heating or Cooling Process
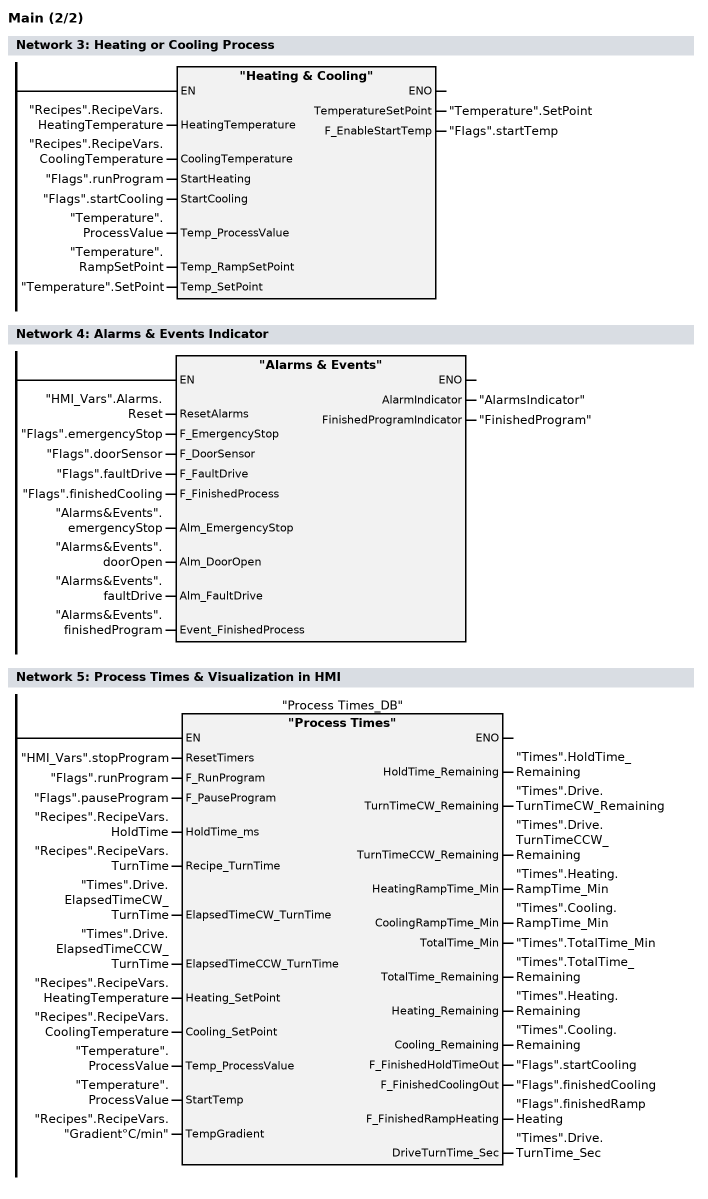
   RUNG wire#powerrail
      "Heating & Cooling"(HeatingTemperature := "Recipes".RecipeVars.HeatingTemperature, CoolingTemperature := "Recipes".RecipeVars.CoolingTemperature, StartHeating := "Flags".runProgram, StartCooling := "Flags".startCooling, Temp_ProcessValue := "Temperature".ProcessValue, Temp_RampSetPoint := "Temperature".RampSetPoint, Temp_SetPoint := "Temperature".SetPoint, TemperatureSetPoint => "Temperature".SetPoint, F_EnableStartTemp => "Flags".startTemp)
   END_RUNG
   // the same network as SCL:
   "Heating & Cooling"(HeatingTemperature := "Recipes".RecipeVars.HeatingTemperature,
                       CoolingTemperature := "Recipes".RecipeVars.CoolingTemperature,
                       StartHeating := "Flags".runProgram,
                       StartCooling := "Flags".startCooling,
                       Temp_ProcessValue := "Temperature".ProcessValue,
                       Temp_RampSetPoint := "Temperature".RampSetPoint,
                       Temp_SetPoint := "Temperature".SetPoint,
                       TemperatureSetPoint => "Temperature".SetPoint,
                       F_EnableStartTemp => "Flags".startTemp);
END_REGION

REGION Network 4: Alarms & Events Indicator
   RUNG wire#powerrail
      "Alarms & Events"(ResetAlarms := "HMI_Vars".Alarms.Reset, F_EmergencyStop := "Flags".emergencyStop, F_DoorSensor := "Flags".doorSensor, F_FaultDrive := "Flags".faultDrive, F_FinishedProcess := "Flags".finishedCooling, Alm_EmergencyStop := "Alarms&Events".emergencyStop, Alm_DoorOpen := "Alarms&Events".doorOpen, Alm_FaultDrive := "Alarms&Events".faultDrive, Event_FinishedProcess := "Alarms&Events".finishedProgram, AlarmIndicator => "AlarmsIndicator", FinishedProgramIndicator => "FinishedProgram")
   END_RUNG
   // the same network as SCL:
   "Alarms & Events"(ResetAlarms := "HMI_Vars".Alarms.Reset,
                     F_EmergencyStop := "Flags".emergencyStop,
                     F_DoorSensor := "Flags".doorSensor,
                     F_FaultDrive := "Flags".faultDrive,
                     F_FinishedProcess := "Flags".finishedCooling,
                     Alm_EmergencyStop := "Alarms&Events".emergencyStop,
                     Alm_DoorOpen := "Alarms&Events".doorOpen,
                     Alm_FaultDrive := "Alarms&Events".faultDrive,
                     Event_FinishedProcess := "Alarms&Events".finishedProgram,
                     AlarmIndicator => "AlarmsIndicator",
                     FinishedProgramIndicator => "FinishedProgram");
END_REGION

REGION Network 5: Process Times & Visualization in HMI
   RUNG wire#powerrail
      "Process Times_DB"(ResetTimers := "HMI_Vars".stopProgram, F_RunProgram := "Flags".runProgram, F_PauseProgram := "Flags".pauseProgram, HoldTime_ms := "Recipes".RecipeVars.HoldTime, Recipe_TurnTime := "Recipes".RecipeVars.TurnTime, ElapsedTimeCW_TurnTime := "Times".Drive.ElapsedTimeCW_TurnTime, ElapsedTimeCCW_TurnTime := "Times".Drive.ElapsedTimeCCW_TurnTime, Heating_SetPoint := "Recipes".RecipeVars.HeatingTemperature, Cooling_SetPoint := "Recipes".RecipeVars.CoolingTemperature, Temp_ProcessValue := "Temperature".ProcessValue, StartTemp := "Temperature".ProcessValue, TempGradient := "Recipes".RecipeVars."Gradient°C/min", HoldTime_Remaining => "Times".HoldTime_Remaining, TurnTimeCW_Remaining => "Times".Drive.TurnTimeCW_Remaining, TurnTimeCCW_Remaining => "Times".Drive.TurnTimeCCW_Remaining, HeatingRampTime_Min => "Times".Heating.RampTime_Min, CoolingRampTime_Min => "Times".Cooling.RampTime_Min, TotalTime_Min => "Times".TotalTime_Min, TotalTime_Remaining => "Times".TotalTime_Remaining, Heating_Remaining => "Times".Heating.Remaining, Cooling_Remaining => "Times".Cooling.Remaining, F_FinishedHoldTimeOut => "Flags".startCooling, F_FinishedCoolingOut => "Flags".finishedCooling, F_FinishedRampHeating => "Flags".finishedRampHeating, DriveTurnTime_Sec => "Times".Drive.TurnTime_Sec)
   END_RUNG
   // the same network as SCL:
   "Process Times_DB"(ResetTimers := "HMI_Vars".stopProgram,   // "Process Times"
                      F_RunProgram := "Flags".runProgram,
                      F_PauseProgram := "Flags".pauseProgram,
                      HoldTime_ms := "Recipes".RecipeVars.HoldTime,
                      Recipe_TurnTime := "Recipes".RecipeVars.TurnTime,
                      ElapsedTimeCW_TurnTime := "Times".Drive.ElapsedTimeCW_TurnTime,
                      ElapsedTimeCCW_TurnTime := "Times".Drive.ElapsedTimeCCW_TurnTime,
                      Heating_SetPoint := "Recipes".RecipeVars.HeatingTemperature,
                      Cooling_SetPoint := "Recipes".RecipeVars.CoolingTemperature,
                      Temp_ProcessValue := "Temperature".ProcessValue,
                      StartTemp := "Temperature".ProcessValue,
                      TempGradient := "Recipes".RecipeVars."Gradient°C/min",
                      HoldTime_Remaining => "Times".HoldTime_Remaining,
                      TurnTimeCW_Remaining => "Times".Drive.TurnTimeCW_Remaining,
                      TurnTimeCCW_Remaining => "Times".Drive.TurnTimeCCW_Remaining,
                      HeatingRampTime_Min => "Times".Heating.RampTime_Min,
                      CoolingRampTime_Min => "Times".Cooling.RampTime_Min,
                      TotalTime_Min => "Times".TotalTime_Min,
                      TotalTime_Remaining => "Times".TotalTime_Remaining,
                      Heating_Remaining => "Times".Heating.Remaining,
                      Cooling_Remaining => "Times".Cooling.Remaining,
                      F_FinishedHoldTimeOut => "Flags".startCooling,
                      F_FinishedCoolingOut => "Flags".finishedCooling,
                      F_FinishedRampHeating => "Flags".finishedRampHeating,
                      DriveTurnTime_Sec => "Times".Drive.TurnTime_Sec);
END_REGION
END_ORGANIZATION_BLOCK

ORGANIZATION_BLOCK "Temperature Control"   // OB30, LAD, CyclicInterrupt
TITLE = PID Temperature Control
{ S7_Optimized_Access := 'TRUE' }
VERSION : 0.1
   VAR_INPUT
      Initial_Call : Bool;   // Initial call of this OB
      Event_Count : Int;   // Events discarded
   END_VAR
BEGIN

REGION Network 1: RTD Format Value, Gradient Temperature and Temperature PID
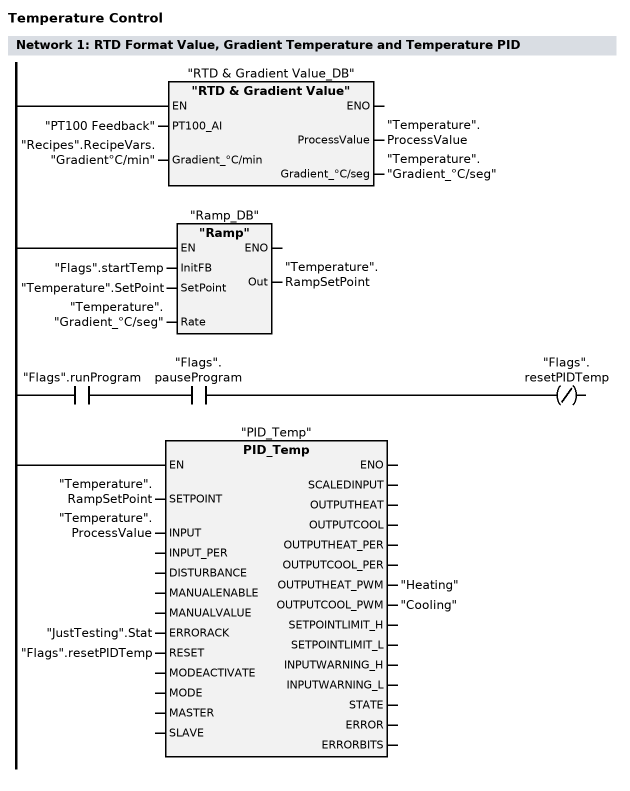
   "RTD & Gradient Value_DB"(PT100_AI := "PT100 Feedback",   // "RTD & Gradient Value"
                           "Gradient_°C/min" := "Recipes".RecipeVars."Gradient°C/min",
                           ProcessValue => "Temperature".ProcessValue,
                           "Gradient_°C/seg" => "Temperature"."Gradient_°C/seg");
   "Ramp_DB"(InitFB := "Flags".startTemp,   // "Ramp"
             SetPoint := "Temperature".SetPoint,
             Rate := "Temperature"."Gradient_°C/seg",
             Out => "Temperature".RampSetPoint);
   "Flags".resetPIDTemp := NOT ("Flags".runProgram AND "Flags".pauseProgram);
   "PID_Temp"(Setpoint := "Temperature".RampSetPoint,   // PID_Temp
              Input := "Temperature".ProcessValue,
              ErrorAck := "JustTesting".Stat,
              Reset := "Flags".resetPIDTemp,
              OutputHeat_PWM => "Heating",
              OutputCool_PWM => "Cooling");
END_REGION
END_ORGANIZATION_BLOCK

(* ===== HMI "HMI_RT_1" =====
system functions are stored by id; their names below are inferred from use
connection "HMI_Connection_1": ETHERNET, SMART_S7_1200_OMS

HMI tags "Tags"
   "Tag_ScreenNumber" : UInt, internal
   "PT100 Feedback" : Int = PLC "PT100 Feedback" AT %IW13, 1 s
   "Temperature_RampSetPoint" : Real = PLC Temperature.RampSetPoint AT %DB4.DBD4, 1 s
   "Recipes_Frequency" : Real = PLC Recipes.RecipeVars.Frequency, 1 s
   "Recipes_HeatingSetPoint" : Real = PLC Recipes.RecipeVars.HeatingTemperature, 1 s
   "Recipes_TurnTime" : DInt = PLC Recipes.RecipeVars.TurnTime, 1 s
   "Recipes_HoldTime" : DInt = PLC Recipes.RecipeVars.HoldTime, 1 s
   "Recipes_Gradient°C/min" : Real = PLC Recipes.RecipeVars.Gradient°C/min, 1 s
   "RTD & Gradient Value_DB_ProcessValue" : Real = PLC "RTD & Gradient Value_DB".ProcessValue, 1 s
   "Temperature_ProcessValue" : Real = PLC Temperature.ProcessValue AT %DB4.DBD8, 1 s
   "HMI_Vars_Drive_handAutoMode" : Bool = PLC HMI_Vars.Drive.handAutoMode, 1 s
   "HMI_Vars_Drive_DriveCW" : Bool = PLC HMI_Vars.Drive.DriveCW, 1 s
   "HMI_Vars_Drive_DriveCCW" : Bool = PLC HMI_Vars.Drive.DriveCCW, 1 s
   "HMI_Vars_Drive_JogCW" : Bool = PLC HMI_Vars.Drive.JogCW, 1 s
   "HMI_Vars_Drive_JogCCW" : Bool = PLC HMI_Vars.Drive.JogCCW, 1 s
   "HMI_Vars_Drive_ResetDrive" : Bool = PLC HMI_Vars.Drive.ResetDrive, 1 s
   "HMI_Vars_Drive_AutoMode" : Bool = PLC HMI_Vars.Drive.AutoMode, 1 s
   "HMI_Vars_Drive_HandMode" : Bool = PLC HMI_Vars.Drive.HandMode, 1 s
   "HMI_Vars_Drive_SetPoint" : Real = PLC HMI_Vars.Drive.SetPoint, 1 s
   "HMI_Vars_Drive_Run" : Bool = PLC HMI_Vars.Drive.Run, 1 s
   "DriveJOGCCW" : Bool = PLC FinishedProgram AT %Q0.3, 1 s
   "DriveJOGCW" : Bool = PLC AlarmsIndicator AT %Q0.2, 1 s
   "Recipes_RecipeName" : String[254] = PLC Recipes.RecipeVars.RecipeName, 1 s
   "HMI_Vars_Alarms_Reset" : Bool = PLC HMI_Vars.Alarms.Reset, 1 s
   "HMI_Vars_runProgram" : Bool = PLC HMI_Vars.runProgram, 1 s
   "AlarmsTrigger" : UInt AT %DB8.DBW0, 1 s
   "AlarmsFlags_faultDrive" : Bool = PLC "Alarms&Events".faultDrive AT %DB8.DBX0.2, 1 s
   "DriveCW" : Bool = PLC DriveCW AT %Q0.0, 1 s
   "DriveCCW" : Bool = PLC DriveCCW AT %Q0.1, 1 s
   "HMI_Vars_stopProgram" : Bool = PLC HMI_Vars.stopProgram, 1 s
   "Times_HoldTime_Remaining" : Real = PLC Times.HoldTime_Remaining, 1 s
   "Times_Drive_TurnTimeCW_Remaining" : Int = PLC Times.Drive.TurnTimeCW_Remaining, 1 s
   "Times_Drive_TurnTimeCCW_Remaining" : Int = PLC Times.Drive.TurnTimeCCW_Remaining, 1 s
   "HMI_Vars_pauseProgram" : Bool = PLC HMI_Vars.pauseProgram, 1 s
   "Times_Temperature_RampTime_Min" : DInt = PLC Times.Heating.RampTime_Min, 1 s
   "Times_Temperature_Remaining" : Real = PLC Times.Heating.Remaining, 1 s
   "Recipes_CoolingSetPoint" : Real = PLC Recipes.RecipeVars.CoolingTemperature, 1 s
   "Times_Cooling_RampTime_Min" : DInt = PLC Times.Cooling.RampTime_Min, 1 s
   "Times_Cooling_Remaining" : Real = PLC Times.Cooling.Remaining, 1 s
   "Times_TotalTime_Min" : Real = PLC Times.TotalTime_Min, 1 s
   "Times_Drive_ElapsedTimeCCW_TurnTime" : Time = PLC Times.Drive.ElapsedTimeCCW_TurnTime, 1 s
   "Flags_startCooling" : Bool = PLC Flags.startCooling, 1 s
   "Flags_runProgram" : Bool = PLC Flags.runProgram, 1 s
   "Flags_finishedRampHeating" : Bool = PLC Flags.finishedRampHeating, 1 s
   "Flags_Drive_CurrentFrequency" : Real = PLC Flags.Drive.CurrentFrequency, 1 s

discrete alarms
   1: 'Paro de Emergencia Activado. Rearme el paro de emergencia. / Paro de Emergencia Activado. Rearme el paro de emergencia.', class Errors, trigger "AlarmsTrigger" bit 8
   2: 'Puerta Abierta. Cierra la puerta para poder iniciar el proceso. / Puerta Abierta. Cierra la puerta para poder iniciar el proceso.', class Warnings, trigger "AlarmsTrigger" bit 9
   3: 'Variador en Falla. Verifique el variador y posteriormente resetear. / Variador en Falla. Verifique el variador y posteriormente resetear.', class Errors, trigger "AlarmsTrigger" bit 10
   4: 'Proceso Finalizado. Presione Reset Eventos Para Reiniciar el Programa. / Proceso Finalizado. Presione Reset Eventos Para Reiniciar el Programa.', class ProgramEvents, trigger "AlarmsTrigger" bit 11

analog alarms
   1: 'Valor de Temperatura Alto.', class Errors, trigger "Temperature_ProcessValue"

recipe "Polyester": Frequency <- "Recipes_Frequency", HeatingTemperature <- "Recipes_HeatingSetPoint", TurnTime <- "Recipes_TurnTime", HoldTime <- "Recipes_HoldTime", Gradient °C/min <- "Recipes_Gradient°C/min", CoolingTemperature <- "Recipes_CoolingSetPoint"

recipe "Nylon": HeatingTemperature <- "Recipes_HeatingSetPoint", CoolingTemperature <- "Recipes_CoolingSetPoint", Gradient °C/min <- "Recipes_Gradient°C/min", Frequency <- "Recipes_Frequency", TurnTime <- "Recipes_TurnTime", HoldTime <- "Recipes_HoldTime"

recipe "Powernet": HeatingTemperature <- "Recipes_HeatingSetPoint", CoolingTemperature <- "Recipes_CoolingSetPoint", Gradient °C/min <- "Recipes_Gradient°C/min", Frequency <- "Recipes_Frequency", TurnTime <- "Recipes_TurnTime", HoldTime <- "Recipes_HoldTime"

Template "Template_1" 480x272
   DateTimeField "HmiScreenItemData" at 395,22 size 85x22
   DateTimeField "HmiScreenItemData_1" at 395,0 size 85x22
   GraphicView "Logo" at 0,0 size 157x38; Picture "Screenshot 2025-11-29 201759"
   Softkey "Softkey_F1" at 0,0 size 0x0
      on KeyUp: ActivateScreen("Root screen", 0)
   Softkey "Softkey_F2" at 0,0 size 0x0
      on KeyUp: ActivateScreen("Buffer Alarms", 0)
   Softkey "Softkey_F3" at 0,0 size 0x0
      on KeyUp: ActivateScreen("System Diagnostics", 0)
   Softkey "Softkey_F4" at 0,0 size 0x0; Authorization "User administration"
      on KeyUp: StopRuntime(0)

screen "Root screen" 480x272, template "Template_1"
   on GenerateScreen: SetTag("Tag_ScreenNumber", 1)
   Button "Template_Button_1" at 17,94 size 94x76; TextOn 'Temperatura'; TextOff 'Temperatura'; PictureOff "query_stats_90dp"
      on Release: ActivateScreen("Temperature Trend View", 0)
   TextField "Template_Text field_1" at 17,57 size 89x52; Text 'Trend Temperatura'
   Button "Template_Button_2" at 133,94 size 94x76; TextOn 'Temperatura'; TextOff 'Temperatura'; PictureOff "recipe"
      on Release: ActivateScreen("Recipes", 0)
   TextField "Template_Text field_2" at 139,58 size 79x36; Text 'Seleccionar Proceso'
   Button "Template_Button_3" at 250,94 size 94x76; TextOn 'Temperatura'; TextOff 'Temperatura'; PictureOff "motion_90dp"
      on Release: ActivateScreen("Drive Control", 0)
   TextField "Template_Text field_3" at 271,58 size 49x36; Text 'Estado Drive'
   TextField "Text field_1" at 207,6 size 147x22; Text 'Rapid Dyeing Machine'
   Button "Button_1" at 367,191 size 97x34; TextOn 'Resseting'; TextOff 'Reset Eventos'; PictureOff "reload"
      on Press: function_b14e0dd5("HMI_Vars_Alarms_Reset", 0)
   Button "Button_2" at 17,191 size 97x34; TextOn 'Running'; TextOff 'Run Program'; PictureOff "reload"
      on Release: SetBit("HMI_Vars_runProgram"); ResetBit("HMI_Vars_stopProgram"); ResetBit("HMI_Vars_pauseProgram")
   Button "Template_Button_6" at 367,94 size 94x76; TextOn 'Temperatura'; TextOff 'Temperatura'; PictureOff "update_200dp"
      on Release: ActivateScreen("Process Times", 0)
   TextField "Template_Text field_6" at 385,58 size 57x36; Text 'Tiempos Proceso'
   Button "Button_3" at 133,191 size 97x34; TextOn 'Paused'; TextOff 'Pause Program'; PictureOff "reload"
      on Release: SetBit("HMI_Vars_pauseProgram")
   Button "Button_4" at 247,191 size 97x34; TextOn 'Stopped'; TextOff 'Stop Program'; PictureOff "reload"
      on Release: SetBit("HMI_Vars_stopProgram"); ResetBit("HMI_Vars_pauseProgram"); ResetBit("HMI_Vars_runProgram")

screen "Temperature Trend View" 480x272, template "Template_1"
   TrendView "Trend view_1" at 1,39 size 477x231
   IOField "I/O field_1" at 214,20 size 63x22; FormatPattern 999.9; Unit °C
      ProcessValue <- "Temperature_RampSetPoint"
   TextField "Text field_1" at 190,20 size 26x22; Text 'SP:'
   IOField "I/O field_2" at 319,20 size 63x22; FormatPattern 999.9; Unit °C
      ProcessValue <- "Temperature_ProcessValue"
   TextField "Text field_2" at 294,20 size 27x22; Text 'PV:'
   TextField "Text field_3" at 190,0 size 47x22; Text 'Batch:'
   IOField "I/O field_3" at 237,1 size 161x22; FormatPattern ???????????
      ProcessValue <- "Recipes_RecipeName"

screen "Recipes" 480x272, template "Template_1"
   RecipeView "Recipe view_1" at 1,39 size 478x232; Tag4RecipeNumber "Recipes_RecipeName"
   TextField "Text field_1" at 170,5 size 47x22; Text 'Batch:'
   IOField "I/O field_3" at 217,6 size 161x22; FormatPattern ???????????
      ProcessValue <- "Recipes_RecipeName"

screen "Drive Control" 480x272, template "Template_1"
   TextField "Text field_1" at 226,11 size 88x22; Text 'Drive Control'
   TextField "Text field_3" at 95,51 size 30x22; Text 'Giro'
   Switch "Switch_1" at 77,80 size 72x28; CaptionText 'Switch'; TextOff 'OFF'; TextOn 'ON'
      ProcessValue <- "HMI_Vars_Drive_DriveCW"
      on SwitchOn: SetBit("HMI_Vars_Drive_DriveCW")
      on SwitchOff: ResetBit("HMI_Vars_Drive_DriveCW")
   GraphicView "Graphic view_1" at 45,85 size 24x24; Picture "reload"
   GraphicView "Graphic view_2" at 45,121 size 24x24; Picture "restore"
   TextField "Text field_4" at 267,49 size 74x22; Text 'Frecuencia'
   TextField "Text field_5" at 38,184 size 79x20; Text 'Drive Status:'
   Circle "Circle_1" at 128,187 size 14x14
      Appearance <- "HMI_Vars_Drive_Run"
   TextField "Text field_6" at 146,184 size 52x20; Text 'Stopped'
      Visibility <- "HMI_Vars_Drive_Run"
   TextField "Text field_7" at 38,206 size 71x20; Text 'Drive Fault:'
   Circle "Circle_2" at 128,209 size 14x14
      Appearance <- "AlarmsFlags_faultDrive"
   TextField "Text field_8" at 147,206 size 47x20; Text 'Healthy'
      Visibility <- "AlarmsFlags_faultDrive"
   TextField "Text field_13" at 234,74 size 111x20; Text 'Frecuencia Actual:'
   IOField "I/O field_1" at 381,74 size 49x20; FormatPattern 99.9; Unit Hz
      ProcessValue <- "Flags_Drive_CurrentFrequency"
   Switch "Switch_2" at 77,119 size 72x28; TextOn 'ON'; CaptionText 'Switch'; TextOff 'OFF'
      ProcessValue <- "HMI_Vars_Drive_DriveCCW"
      on SwitchOn: SetBit("HMI_Vars_Drive_DriveCCW")
      on SwitchOff: ResetBit("HMI_Vars_Drive_DriveCCW")
   TextField "Text field_16" at 152,207 size 33x20; Text 'Fault'
      Visibility <- "AlarmsFlags_faultDrive"
   TextField "Text field_17" at 38,229 size 74x20; Text 'Drive Mode:'
   Circle "Circle_5" at 128,232 size 14x14
      Appearance <- "HMI_Vars_Drive_AutoMode"
   TextField "Text field_18" at 149,229 size 31x20; Text 'Auto'
      Visibility <- "HMI_Vars_Drive_AutoMode"
   TextField "Text field_19" at 153,230 size 34x20; Text 'Hand'
      Visibility <- "HMI_Vars_Drive_HandMode"
   TextField "Text field_20" at 147,185 size 51x20; Text 'Running'
      Visibility <- "HMI_Vars_Drive_Run"
   TextField "Text field_21" at 234,128 size 97x20; Text 'Manual SetPoint'
   TextField "Text field_22" at 242,198 size 63x20; Text 'Drive CW:'
   Circle "Circle_6" at 340,201 size 14x14
      Appearance <- "DriveCW"
   TextField "Text field_23" at 358,198 size 46x20; Text 'Disable'
      Visibility <- "DriveCW"
   TextField "Text field_24" at 359,198 size 43x20; Text 'Enable'
      Visibility <- "DriveCW"
   TextField "Text field_25" at 242,221 size 71x20; Text 'Drive CCW:'
   Circle "Circle_7" at 340,224 size 14x14
      Appearance <- "DriveCCW"
   TextField "Text field_26" at 358,221 size 46x20; Text 'Disable'
      Visibility <- "DriveCCW"
   TextField "Text field_27" at 362,221 size 43x20; Text 'Enable'
      Visibility <- "DriveCCW"
   IOField "I/O field_3" at 357,123 size 66x29; FormatPattern 99.9
      ProcessValue <- "HMI_Vars_Drive_SetPoint"
   TextField "Text field_2" at 234,96 size 123x20; Text 'Frecuencia SetPoint:'
   IOField "I/O field_2" at 381,96 size 49x20; FormatPattern 99.9; Unit Hz
      ProcessValue <- "Recipes_Frequency"

screen "System Diagnostics" 480x272, template "Template_1"
   SysDiagControl "System diagnostics view_1" at 1,39 size 476x232
   TextField "Text field_1" at 201,7 size 131x22; Text 'System Diagnostics'

screen "Maintenance" 480x272, template "Template_1"
   TextField "Text field_1" at 226,11 size 87x22; Text 'Maintenance'
   Button "Button_1" at 114,122 size 85x30; TextOn 'Stopped'; TextOff 'Stop PLC'; PictureOff "reload"; Authorization "User administration"
      on Release: function_f249594b("HMI_Connection_1", 4)
   Button "Button_2" at 226,122 size 85x30; TextOn 'Running'; TextOff 'Run PLC'; PictureOff "reload"
      on Release: function_f249594b("HMI_Connection_1", 8)

screen "Buffer Alarms" 480x272, template "Template_1"
   AlarmView "Alarm view_1" at 1,40 size 477x230
   TextField "Text field_1" at 181,8 size 202x22; Text 'Historial de Alarmas y Eventos'

screen "Process Times" 480x272, template "Template_1"
   TextField "Text field_1" at 205,10 size 138x22; Text 'Tiempos de Proceso'
   IOField "I/O field_1" at 179,62 size 42x20; FormatPattern 999; Unit m
      ProcessValue <- "Recipes_HoldTime"
   TextField "Text field_2" at 26,60 size 100x22; Text 'Sostenimiento:'
   IOField "I/O field_2" at 177,85 size 58x20; FormatPattern 999.9; Unit m
      ProcessValue <- "Times_HoldTime_Remaining"
   TextField "Text field_3" at 27,83 size 139x22; Text 'Rest. Sostenimiento:'
   IOField "I/O field_3" at 181,121 size 30x20; FormatPattern 99; Unit s
      ProcessValue <- "Recipes_TurnTime"
   TextField "Text field_4" at 27,119 size 78x22; Text 'Giro Motor:'
   IOField "I/O field_4" at 181,143 size 30x20; FormatPattern 99; Unit s
      ProcessValue <- "Times_Drive_TurnTimeCW_Remaining"
   TextField "Text field_5" at 27,141 size 145x22; Text 'Rest. Giro Motor CW:'
   IOField "I/O field_5" at 398,62 size 34x20; FormatPattern 99; Unit m
      ProcessValue <- "Times_Temperature_RampTime_Min"
   TextField "Text field_6" at 272,60 size 110x22; Text 'Rampa Heating:'
   IOField "I/O field_6" at 396,85 size 50x20; FormatPattern 99.9; Unit m
      ProcessValue <- "Times_Temperature_Remaining"
   TextField "Text field_7" at 273,83 size 95x22; Text 'Rest. Rampa:'
   IOField "I/O field_7" at 397,122 size 34x20; FormatPattern 99; Unit m
      ProcessValue <- "Times_Cooling_RampTime_Min"
   TextField "Text field_8" at 271,120 size 106x22; Text 'Rampa Cooling:'
   IOField "I/O field_8" at 395,145 size 50x20; FormatPattern 99.9; Unit m
      ProcessValue <- "Times_Cooling_Remaining"
   TextField "Text field_9" at 272,143 size 95x22; Text 'Rest. Rampa:'
   IOField "I/O field_9" at 271,212 size 58x20; FormatPattern 999.9; Unit m
      ProcessValue <- "Times_TotalTime_Min"
   TextField "Text field_10" at 107,210 size 97x22; Text 'Tiempo Total:'
   IOField "I/O field_10" at 181,167 size 30x20; FormatPattern 99; Unit s
      ProcessValue <- "Times_Drive_TurnTimeCCW_Remaining"
   TextField "Text field_11" at 27,165 size 154x22; Text 'Rest. Giro Motor CCW:'
   Circle "Circle_5" at 9,75 size 14x14
      Appearance <- "Flags_finishedRampHeating"
      Visibility <- "Flags_finishedRampHeating"
   Circle "Circle_1" at 252,75 size 14x14
      Appearance <- "Flags_runProgram"
      Visibility <- "Flags_runProgram"
   Circle "Circle_2" at 252,138 size 14x14
      Appearance <- "Flags_startCooling"
      Visibility <- "Flags_startCooling"
*)